// TwinCAT 3 PLC project Plc
// ProgramVersion: 3.1.4024.0
// libraries:
//   Tc2_MC2, * (Beckhoff Automation GmbH)
//   Tc2_Standard, * (Beckhoff Automation GmbH)
//   Tc2_System, * (Beckhoff Automation GmbH)
//   Tc3_Module, * (Beckhoff Automation GmbH)
//   VisuSymbols,3.5.10.0,System
// project tree:
//   / Gestore di visualizzazione.TcVMO (not stored), GlobalTextList.TcGTLO, PlcTask.TcTTO
//   GVLs/ Gvl.TcGVL
//   POUs/ MAIN.TcPOU
//   VISUs/ Visualization.TcVIS
// real-time tasks:
//   TASK PlcTask: cycle T#10ms, priority 20, ADS port 350
// motion (NC):
//   TASK NC-Task 1 SAF: cycle T#2ms, priority 4, ADS port 501
//   TASK NC-Task 1 SVB: cycle T#10ms, priority 8, ADS port 511
//   AXIS Asse 1 (id 1)
//     OtherSettings: AllowMotionCmdToSlave=true
//     encoder EncType=1
//     drive DrvType=5
//       Analog: TorqueSetpointScale=10, ScaleFactorActTorque=0.1
//     controller CtrType=1
//       CtrPara: PriorControlFactor=1
//         Observer: BandWidth=20
// variable links:
//   Plc/Plc Instance <-> NC-Task 1 SAF/Axes/Asse 1
//     PlcTask Inputs/Gvl.Axis.NcToPlc <-> Outputs/ToPlc
//     PlcTask Outputs/Gvl.Axis.PlcToNc <-> Inputs/FromPlc

CONFIGURATION Plc
    RESOURCE PLC ON TwinCAT3
        TASK PlcTask(INTERVAL := T#10ms, PRIORITY := 20);
        PROGRAM MAIN WITH PlcTask : MAIN;
    END_RESOURCE
END_CONFIGURATION

// ---- GVLs/Gvl.TcGVL
{attribute 'qualified_only'}
VAR_GLOBAL
	Axis: AXIS_REF;
	PbStart: BOOL;
	PbStop: BOOL;
END_VAR

// ---- POUs/MAIN.TcPOU
PROGRAM MAIN
VAR
	Power: MC_Power;
	MoveVelocity: MC_MoveVelocity;
	Halt: MC_Halt;
	ReadStatus: MC_ReadStatus;
	Timer: TON;
END_VAR

StartStopMotor();

ACTION StartStopMotor:
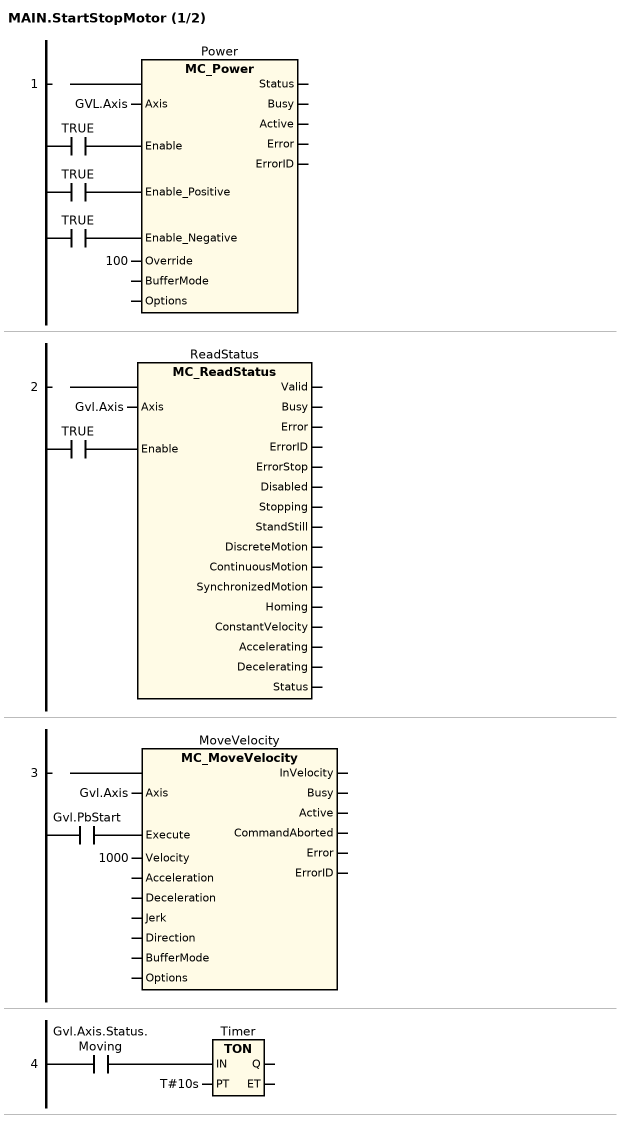
// NETWORK 1
Power(Axis := GVL.Axis, Enable := TRUE, Enable_Positive := TRUE, Enable_Negative := TRUE, Override := 100); // MC_Power

// NETWORK 2
ReadStatus(Axis := Gvl.Axis, Enable := TRUE); // MC_ReadStatus

// NETWORK 3
MoveVelocity(Axis := Gvl.Axis, Execute := Gvl.PbStart, Velocity := 1000); // MC_MoveVelocity

// NETWORK 4
Timer(IN := Gvl.Axis.Status.Moving, PT := T#10s); // TON

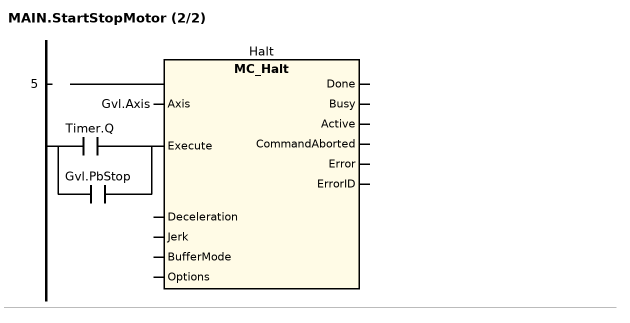
// NETWORK 5
Halt(Axis := Gvl.Axis, Execute := Timer.Q OR Gvl.PbStop); // MC_Halt
END_ACTION

END_PROGRAM

// ---- GlobalTextList.TcGTLO
TEXTLIST GlobalTextList
  170 = 'Motore in movimento'
  314 = 'Start'
  586 = 'Stop'
  146 = 'Testo'
END_TEXTLIST

// ---- VISUs/Visualization.TcVIS
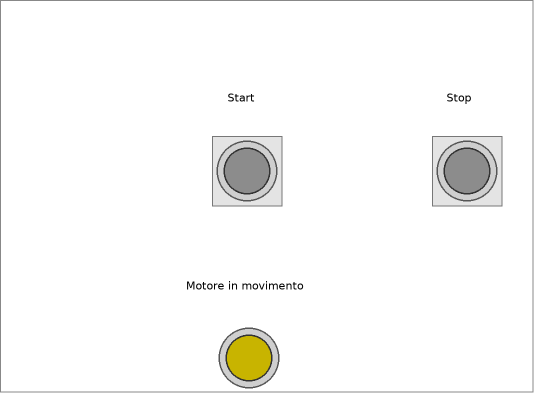
VISUALIZATION Visualization  // 534x393
    PushSwitch (212,136 70x70), variable: Gvl.PbStart, behaviour: TAP, style: Switch-PushSwitch-Gray
    PushSwitch (432,136 70x70), variable: Gvl.PbStop, behaviour: TAP, style: Switch-PushSwitch-Gray
    Label (166,83 150x30), "Start"
    Label (384,83 150x30), "Stop"
    Lamp1 (214,323 70x70), variable: Gvl.Axis.Status.Moving, style: Lamp-Lamp1-Yellow
    Label (170,271 150x30), "Motore in movimento"
END_VISUALIZATION
